Xinje XCPPro project, PLC1: XC3-24 (software 3.3L)

PROGRAM Ladder

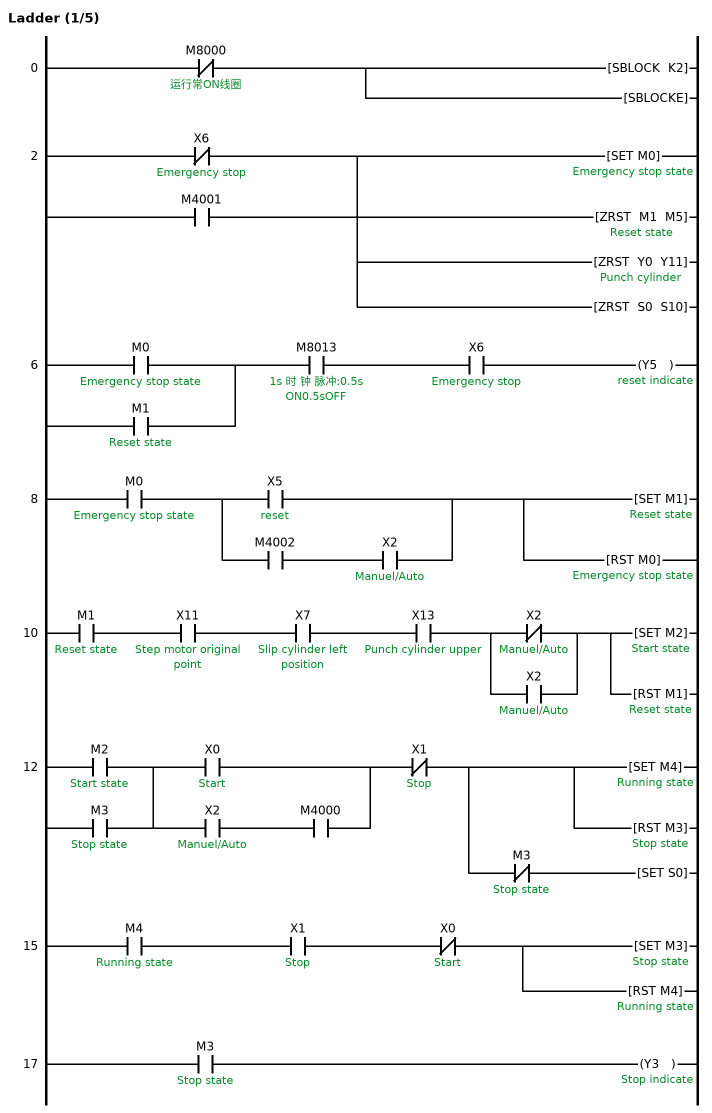
LDI    M8000	; 运行常ON线圈
SBLOCK K2
SBLOCKE
LDI    X6	; Emergency stop
OR     M4001
SET    M0	; Emergency stop state
ZRST   M1 M5	; Reset state
ZRST   Y0 Y11	; Punch cylinder
ZRST   S0 S10
LD     M0	; Emergency stop state
OR     M1	; Reset state
AND    M8013	; 1s 时 钟 脉冲:0.5s ON0.5sOFF
AND    X6	; Emergency stop
OUT    Y5	; reset indicate
LD     M0	; Emergency stop state
LD     X5	; reset
LD     M4002
AND    X2	; Manuel/Auto
ORB
ANB
SET    M1	; Reset state
RST    M0	; Emergency stop state
LD     M1	; Reset state
AND    X11	; Step motor original point
AND    X7	; Slip cylinder left position
AND    X13	; Punch cylinder upper
LDI    X2	; Manuel/Auto
OR     X2	; Manuel/Auto
ANB
SET    M2	; Start state
RST    M1	; Reset state
LD     M2	; Start state
OR     M3	; Stop state
LD     X0	; Start
LD     X2	; Manuel/Auto
AND    M4000
ORB
ANB
ANI    X1	; Stop
SET    M4	; Running state
RST    M3	; Stop state
ANI    M3	; Stop state
SET    S0
LD     M4	; Running state
AND    X1	; Stop
ANI    X0	; Start
SET    M3	; Stop state
RST    M4	; Running state
LD     M3	; Stop state
OUT    Y3	; Stop indicate

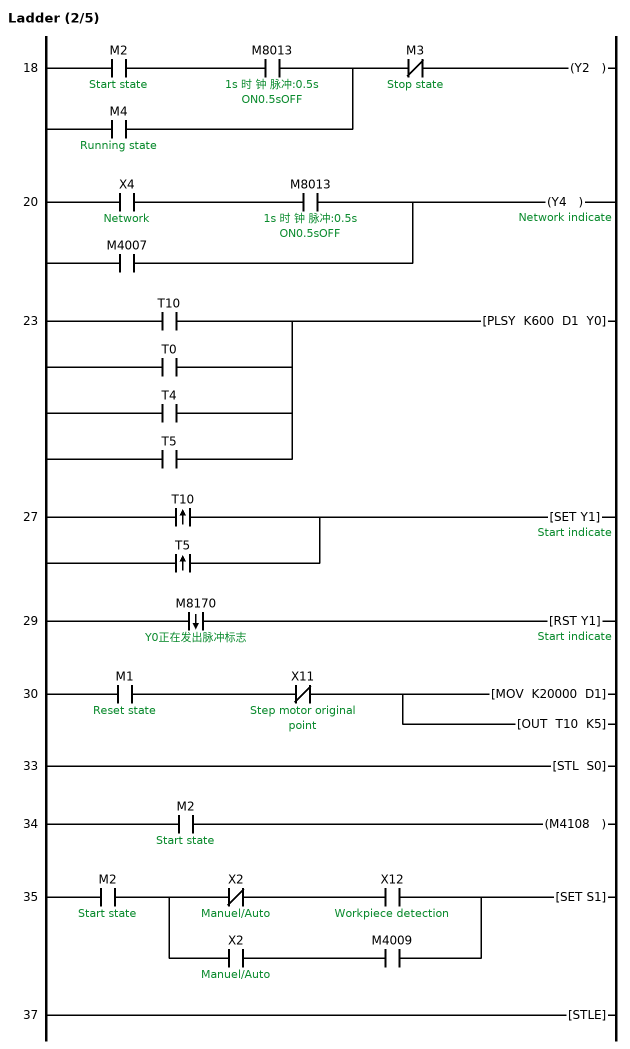
LD     M2	; Start state
AND    M8013	; 1s 时 钟 脉冲:0.5s ON0.5sOFF
OR     M4	; Running state
ANI    M3	; Stop state
OUT    Y2
LD     X4	; Network
AND    M8013	; 1s 时 钟 脉冲:0.5s ON0.5sOFF
OR     M4007
OUT    Y4	; Network indicate
LD     T10
OR     T0
OR     T4
OR     T5
PLSY   K600 D1 Y0
LDP    T10
ORP    T5
SET    Y1	; Start indicate
LDF    M8170	; Y0正在发出脉冲标志
RST    Y1	; Start indicate
LD     M1	; Reset state
ANI    X11	; Step motor original point
MOV    K20000 D1
OUT    T10 K5
STL    S0
LD     M2	; Start state
OUT    M4108
LD     M2	; Start state
LDI    X2	; Manuel/Auto
AND    X12	; Workpiece detection
LD     X2	; Manuel/Auto
AND    M4009
ORB
ANB
SET    S1
STLE

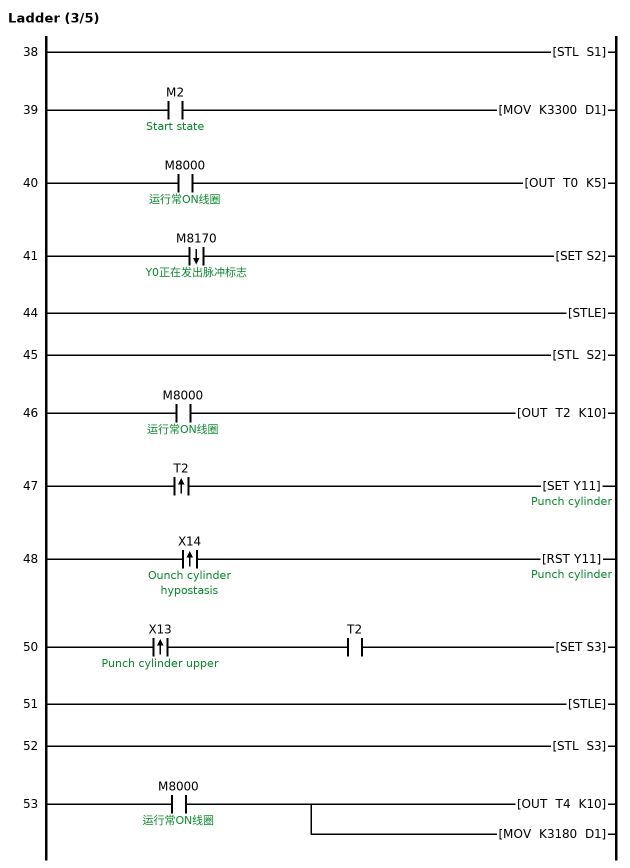
STL    S1
LD     M2	; Start state
MOV    K3300 D1
LD     M8000	; 运行常ON线圈
OUT    T0 K5
LDF    M8170	; Y0正在发出脉冲标志
SET    S2
STLE
STL    S2
LD     M8000	; 运行常ON线圈
OUT    T2 K10
LDP    T2
SET    Y11	; Punch cylinder
LDP    X14	; Ounch cylinder hypostasis
RST    Y11	; Punch cylinder
LDP    X13	; Punch cylinder upper
AND    T2
SET    S3
STLE
STL    S3
LD     M8000	; 运行常ON线圈
OUT    T4 K10
MOV    K3180 D1

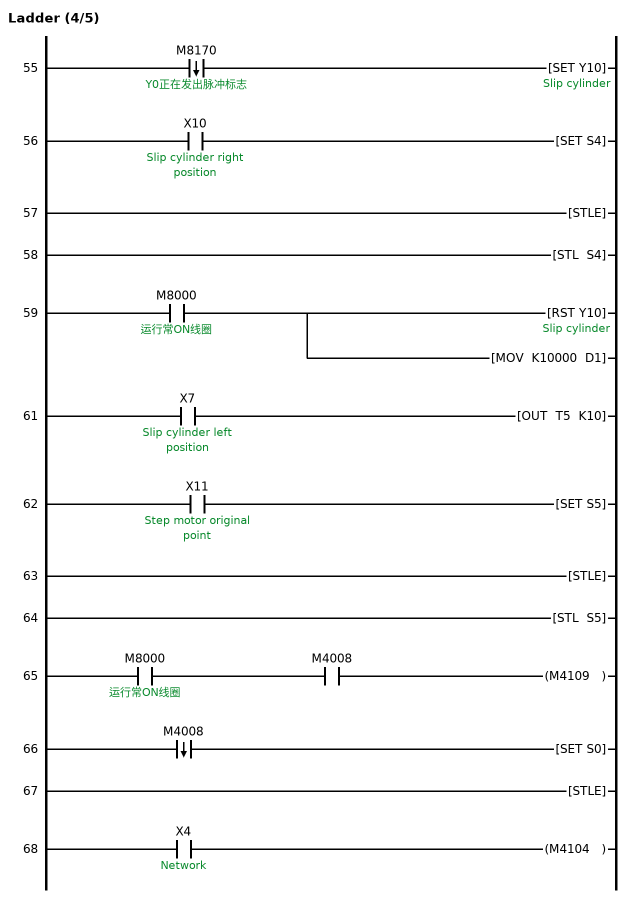
LDF    M8170	; Y0正在发出脉冲标志
SET    Y10	; Slip cylinder
LD     X10	; Slip cylinder right position
SET    S4
STLE
STL    S4
LD     M8000	; 运行常ON线圈
RST    Y10	; Slip cylinder
MOV    K10000 D1
LD     X7	; Slip cylinder left position
OUT    T5 K10
LD     X11	; Step motor original point
SET    S5
STLE
STL    S5
LD     M8000	; 运行常ON线圈
AND    M4008
OUT    M4109
LDF    M4008
SET    S0
STLE
LD     X4	; Network
OUT    M4104

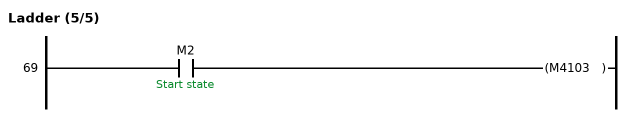
LD     M2	; Start state
OUT    M4103

COMMENTS (devices not used above)
Y6	Alarm indicate